// TIA Portal V20 export
DATA_BLOCK "Alarms"   // DB60
// stored: MemoryReserve 100, Namespace Unit1.Em6
   VAR
      emAlarms { ExternalWritable := 'False'} : "LAF_typeAlarms";
      maintenanceFaults { ExternalWritable := 'False'} : Array[0..199] of Bool;   // PFE Maintenance Faults
      productionFaults { ExternalWritable := 'False'} : Array[0..199] of Bool;   // PFE Production Faults
      toolingFault { ExternalWritable := 'False'} : Array[0..199] of Bool;   // PFE Tooling Faults
      qualityFault { ExternalWritable := 'False'} : Array[0..199] of Bool;   // PFE Quality Faults
      throughputFaultBlocked { ExternalWritable := 'False'} : Array[0..199] of Bool;   // PFE Throughput Fault Blocked
      throughputFaultStarved { ExternalWritable := 'False'} : Array[0..199] of Bool;   // PFE Throughput Fault Starved
      throughputFault { ExternalWritable := 'False'} : Array[0..199] of Bool;   // PFE Throughput Fault
      systemFaultGeneral { ExternalWritable := 'False'} : Array[0..199] of Bool;   // PFE System Fault General
      materialFault { ExternalWritable := 'False'} : Array[0..199] of Bool;   // PFE Material Fault
      maintenanceWarnings { ExternalWritable := 'False'} : Array[0..199] of Bool;   // PFE Maintenance Warnings
      productionWarning { ExternalWritable := 'False'} : Array[0..199] of Bool;   // PFE Production Warning
      toolingWarning { ExternalWritable := 'False'} : Array[0..199] of Bool;   // PFE Tooling Warning
      qualityWarning { ExternalWritable := 'False'} : Array[0..199] of Bool;   // PFE Quality Warning
      throughputWarning { ExternalWritable := 'False'} : Array[0..199] of Bool;   // PFE Throughput Warning
      systemWarning { ExternalWritable := 'False'} : Array[0..199] of Bool;   // PFE System Warning
      materialWarning { ExternalWritable := 'False'} : Array[0..199] of Bool;   // PFE Material Warning
      maintenanceStatus { ExternalWritable := 'False'} : Array[0..199] of Bool;   // PFE Maintenance Status
      productionStatus { ExternalWritable := 'False'} : Array[0..199] of Bool;   // PFE Production Status
      toolingStatus { ExternalWritable := 'False'} : Array[0..199] of Bool;   // PFE Tooling Status
      qualityStatus { ExternalWritable := 'False'} : Array[0..199] of Bool;   // PFE Quality Status
      throughputStatus { ExternalWritable := 'False'} : Array[0..199] of Bool;   // PFE Throughput Status
      systemStatus { ExternalWritable := 'False'} : Array[0..199] of Bool;   // PFE System Status
      materialStatus { ExternalWritable := 'False'} : Array[0..199] of Bool;   // PFE Material Status
      tonMaintenanceFault { ExternalWritable := 'False'} : Array[0..199] of TON_TIME;   // PFE Maintenance Faults Ton Timer
      tonProductionFault { ExternalWritable := 'False'} : Array[0..199] of TON_TIME;   // PFE Production Faults Ton Timer
      tonToolingFault { ExternalWritable := 'False'} : Array[0..199] of TON_TIME;   // PFE Tooling Faults Ton Timer
      tonQualityFault { ExternalWritable := 'False'} : Array[0..199] of TON_TIME;   // PFE Quality Faults Ton Timer
      tonThroughputFaultBlocked { ExternalWritable := 'False'} : Array[0..199] of TON_TIME;   // PFE Throughput Fault Blocked Ton Timer
      tonThroughputFaultStarved { ExternalWritable := 'False'} : Array[0..199] of TON_TIME;   // PFE Throughput Fault Starved Ton Timer
      tonThroughputFault { ExternalWritable := 'False'} : Array[0..199] of TON_TIME;   // PFE Throughput Fault Ton Timer
      tonSystemFaultGeneral { ExternalWritable := 'False'} : Array[0..199] of TON_TIME;   // PFE System Fault General Ton Timer
      tonMaterialFault { ExternalWritable := 'False'} : Array[0..199] of TON_TIME;   // PFE Material Fault Ton Timer
      tonMaintenanceWarning { ExternalWritable := 'False'} : Array[0..199] of TON_TIME;   // PFE Maintenance Warnings Ton Timer
      tonProductionWarning { ExternalWritable := 'False'} : Array[0..199] of TON_TIME;   // PFE Production Warning Ton Timer
      tonToolingWarning { ExternalWritable := 'False'} : Array[0..199] of TON_TIME;   // PFE Tooling Warning Ton Timer
      tonQualityWarning { ExternalWritable := 'False'} : Array[0..199] of TON_TIME;   // PFE Quality Warning Ton Timer
      tonThroughputWarning { ExternalWritable := 'False'} : Array[0..199] of TON_TIME;   // PFE Throughput Warning Ton Timer
      tonSystemWarning { ExternalWritable := 'False'} : Array[0..199] of TON_TIME;   // PFE System Warning Ton Timer
      tonMaterialWarning { ExternalWritable := 'False'} : Array[0..199] of TON_TIME;   // PFE Material Warning Ton Timer
      tonMaintenanceStatus { ExternalWritable := 'False'} : Array[0..199] of TON_TIME;   // PFE Maintenance Status Ton Timer
      tonProductionStatus { ExternalWritable := 'False'} : Array[0..199] of TON_TIME;   // PFE Production Status Ton Timer
      tonToolingStatus { ExternalWritable := 'False'} : Array[0..199] of TON_TIME;   // PFE Tooling Status Ton Timer
      tonQualityStatus { ExternalWritable := 'False'} : Array[0..199] of TON_TIME;   // PFE Quality Status Ton Timer
      tonThroughputStatus { ExternalWritable := 'False'} : Array[0..199] of TON_TIME;   // PFE Throughput Status Ton Timer
      tonSystemStatus { ExternalWritable := 'False'} : Array[0..199] of TON_TIME;   // PFE System Status Ton Timer
      tonMaterialStatus { ExternalWritable := 'False'} : Array[0..199] of TON_TIME;   // PFE Material Status Ton Timer
   END_VAR
BEGIN
   // maintenanceFaults[1] : Hot Press Left Servo Press
END_DATA_BLOCK
